FUNCTION_BLOCK Damper EXTENDS BaseDamper
VAR_INPUT
	IO_Open: REFERENCE TO DigitalOutput;
	IO_FB1, IO_FB2: REFERENCE TO DigitalInput;
END_VAR
VAR_OUTPUT
END_VAR
VAR
	DamperMonitor: DamperMonitor; 
	Error: BOOL;
END_VAR

DamperMonitor(Damper := Open, FB1 := IsOpen, FB2 := IsClosed);
Error := DamperMonitor.Error;

END_FUNCTION_BLOCK

(* stored: Version 1.1.0.1, ProductVersion 3.1.4024.3
   POU Damper: Id {fab3892b-c50d-4312-9c0b-fc77bd04201c}, SpecialFunc None *)
